SUBAPPLICATION Reset (* Subapplication Type *)
  (* Standard: 61499-2 *)
  (* Version 1.0, 2023-02-17, Franz *)
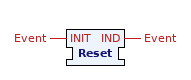
  EVENT_INPUT
    INIT;
  END_EVENT
  EVENT_OUTPUT
    IND;
  END_EVENT
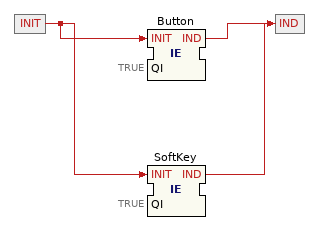
  FBS
    Button : IE(QI := TRUE);
    SoftKey : IE(QI := TRUE);
  END_FBS
  EVENT_CONNECTIONS
    INIT TO Button.INIT;
    Button.IND TO IND;
    INIT TO SoftKey.INIT;
    SoftKey.IND TO IND;
  END_CONNECTIONS
END_SUBAPPLICATION
